{attribute 'qualified_only'}
{attribute 'strict'}
TYPE E_Trend_VISU_Type :
(
	E_VISU_800_480 := 0,
	E_VISU_4_3 :=1
);
END_TYPE

(* stored: Version 1.1.0.1, ProductVersion 3.1.4022.11
   DUT E_Trend_VISU_Type: Id {ddf33f10-9079-4a66-9529-38ddc547ef5f} *)
